// Mitsubishi GX Works2 project: 18   PLC: FX3G

// task Task_01 (event TRUE, interval 0, priority 31): POU_01

PROGRAM POU_01
VAR
  wstep : INT;
  ton1 : TON;
  cnt : INT;
END_VAR
IF M8002 THEN
	wstep := 0;
END_IF;

IF NOT M0 THEN
	wstep := 0;
END_IF;

CASE wstep OF
	0:
		zrst(TRUE, Y0, Y3);
		
		IF M0 THEN
			wstep := 20;
		END_IF;

	20:
		ton1(in := NOT ton1.q, pt := t#3s);
		Z0 := cnt;
		IF ton1.q THEN
			cnt := cnt + 1;
			cnt := cnt MOD 3;
		END_IF;
		zrst(TRUE, Y0, Y3);
		Y0Z0 := M8013;
		
		IF M1 THEN
			wstep := 30;
		END_IF;
		
	30:
		Y2 := M8013;
		
		IF NOT M1 THEN
			wstep := 20;
		END_IF;
END_CASE;
END_PROGRAM
